# EPICS autosave request: iocBoot/ioc13idc_linux/auto_positions.req
file "Galil_positions.req", P=$(P)
file "XPS_positions.req",   P=$(P)
